FUNCTION_BLOCK FB_FrmWcStateDiagnosis
VAR_OUTPUT
	bError						:BOOL;								//エラー発生を出力
END_VAR
VAR
	uiFrmWcState 		AT%I*	:UINT;								//PDデータとリンク
	
	bErrorState					:ARRAY[0..15] OF BOOL;				//各ステートエラー
	fbBitREdge					:ARRAY[0..15] OF R_TRIG;
	bSendMsgMem					:ARRAY[0..14] OF BOOL;				//メッセージ送信を記憶	
	sSendMsgString				:STRING;							//送信メッセージのアーギュメント用
	bSendMsg					:BOOL;								//メッセージ送信予約
	fbMessage					:ARRAY[0..1] OF FB_TcMessage;
	i							:INT;
END_VAR

//エラー状態を出力
	bError:= uiFrmWcState<>0 ;
	
//サイクリックフレームごとのワーキングカウンターチェック、エラーは複数発生する可能性があるので全bitチェック
	FOR i := 0 TO 15 DO
		bErrorState[i]:=(uiFrmWcState AND SHL(1,i))<>0;
	END_FOR
	
//結果をEventloggerへ
	bSendMsg:=FALSE;	//メッセージ送信予約をリセット

	FOR i := 0 TO 14 BY 1 DO
		//エラーの立ち上がりエッジを検出
		fbBitREdge[i](CLK:=bErrorState[i]);
		
		//まだ送信していなければ、送信用の文字列作成
		IF NOT bSendMsgMem[i] AND fbBitREdge[i].Q THEN
			
			sSendMsgString:=CONCAT(sSendMsgString, CONCAT(INT_TO_STRING(i+1), '. '));	//送信メッセージのアーギュメント作成

			bSendMsg:=TRUE;		//メッセージ送信予約をセット
			bSendMsgMem[i]:=TRUE;	//メッセージ送信を記憶
			
		END_IF
		
		//エラーがリセットされたらメッセージ送信気を記憶をリセット
		IF NOT bErrorState[i] THEN
			bSendMsgMem[i]:=FALSE;
		END_IF
		
	END_FOR
	
	IF bSendMsg THEN
		fbMessage[0].ipArguments.Clear().AddString(sSendMsgString);
		fbMessage[0].Send();
		
		bSendMsg:=FALSE;
		sSendMsgString:='';
	END_IF
	
	//全体判定用
	fbBitREdge[15](CLK:=bErrorState[15]);
	
	IF fbBitREdge[15].Q THEN
		fbMessage[1].Send();
	END_IF

//FB_Init は常に暗黙的に使用可能で、主に初期化に使用されます。
//戻り値は評価されません。特定の結果を得るために、メソッドを明示的に宣言し、
//そのメソッドに標準の初期化コードをもったコードを追加することができます。戻り値を評価できます。
METHOD FB_Init: BOOL
VAR_INPUT
    bInitRetains: BOOL; // TRUE: 保持変数は初期化されます (ウォーム リセット、あるいはコールド リセット)
    bInCopyCode: BOOL;  // TRUE: 後でコードをコピーする (オンライン変更) ために、インスタンスをコピーします。
END_VAR
fbMessage[0].CreateEx(TC_EVENTS.TkEtherCATMasterDiagnosisEventClass.WrongWorkingCounterEtherCATCommandReceived);
fbMessage[1].CreateEx(TC_EVENTS.TkEtherCATMasterDiagnosisEventClass.CompleteFrameMissing);
END_METHOD

END_FUNCTION_BLOCK

(* stored: Version 1.1.0.1, ProductVersion 3.1.4026.18
   POU FB_FrmWcStateDiagnosis: Id {4e91cd08-8953-4bd4-ae28-be45cc439d43}, SpecialFunc None
   Method FB_Init: Id {7a56f216-0586-4f04-a2eb-3842cf2c6d30} *)
